// TIA Portal project "ASSEMBLER" (V16)

(* hardware
DEVICE "S7300/ET200M station_1"  S7-300 station
   slot 0: "Rail_0"  Rail  6ES7 390-1***0-0AA0
   slot 2: "PLC_1"  CPU 313C  6ES7 313-5BF03-0AB0  V2.6
      slot 0: "MPI interface_1"  X1
      slot 2: "DI 24/DO 16_1"  DI24/DO16
      slot 3: "AI 5/AO 2_1"  AI5/AO2
      slot 4: "Count_1"  Counter
*)

// ===== PLC "PLC_1"  CPU 313C =====

VAR_GLOBAL   // PLC tag table "Default tag table"
   "MOVING X" AT %I0.0 : Bool;
   "MOVING Z" AT %I0.1 : Bool;
   "ITEM DETECTED" AT %I0.2 : Bool;
   "LID AT PLACE" AT %I0.3 : Bool;
   "LID CLAMPED" AT %I0.4 : Bool;
   "POS.AT LIMIT(LIDS)" AT %I0.5 : Bool;
   "BASE AT PLACE" AT %I0.6 : Bool;
   "BASE CLAMPED" AT %I0.7 : Bool;
   "POS. AT LIMIT(BASES)" AT %I1.0 : Bool;
   "PART LEAVING" AT %I1.1 : Bool;
   "START" AT %I1.2 : Bool;
   "RESET" AT %I1.3 : Bool;
   "STOP" AT %I1.4 : Bool;
   "EMERGENCY" AT %I1.5 : Bool;
   "AUTO" AT %I1.6 : Bool;
   "MOVE X" AT %Q0.0 : Bool;
   "MOVE Z" AT %Q0.1 : Bool;
   "GRAB" AT %Q0.2 : Bool;
   "LIDS CONVEYOR" AT %Q0.3 : Bool;
   "CLAMP LID" AT %Q0.4 : Bool;
   "POS. RAISE(LID)" AT %Q0.5 : Bool;
   "BASES CONVEYOR" AT %Q0.6 : Bool;
   "CLAMP BASE" AT %Q0.7 : Bool;
   "POS. RAISE (BASES)" AT %Q1.0 : Bool;
   "START LIGHT" AT %Q1.1 : Bool;
   "RESET LIGHT" AT %Q1.2 : Bool;
   "STOP LIGHT" AT %Q1.3 : Bool;
   "COUNTER" AT %QD30 : DInt;
   "M_LID AT PLACE" AT %M0.0 : Bool;
   "stop_lid_conveyor" AT %M0.1 : Bool;
   "m_base at place" AT %M0.2 : Bool;
   "stop_base_conveyor" AT %M0.3 : Bool;
   "m_z" AT %M0.4 : Bool;
   "Run_grab" AT %M0.5 : Bool;
   "m_x" AT %M0.6 : Bool;
   "Run_x" AT %M0.7 : Bool;
   "Tag_1" AT %M1.0 : Bool;
   "set_z_after_x" AT %M1.1 : Bool;
   "Tag_2" AT %M1.2 : Bool;
   "reset grab_after x" AT %M1.3 : Bool;
   "Tag_3" AT %M1.4 : Bool;
   "set again base conveyor" AT %M1.5 : Bool;
   "Tag_4" AT %M1.6 : Bool;
   "reset system" AT %M1.7 : Bool;
   "NUMBER" AT %MD2 : DInt;
END_VAR

ORGANIZATION_BLOCK "Main"   // OB1, STL
TITLE = "Main Program Sweep (Cycle)"
{ S7_Optimized_Access := 'FALSE' }
VERSION : 0.1
   VAR_TEMP
      OB1_EV_CLASS : Byte;   // Bits 0-3 = 1 (Coming event), Bits 4-7 = 1 (Event class 1)
      OB1_SCAN_1 : Byte;   // 1 (Cold restart scan 1 of OB 1), 3 (Scan 2-n of OB 1)
      OB1_PRIORITY : Byte;   // Priority of OB Execution
      OB1_OB_NUMBR : Byte;   // 1 (Organization block 1, OB1)
      OB1_RESERVED_1 : Byte;   // Reserved for system
      OB1_RESERVED_2 : Byte;   // Reserved for system
      OB1_PREV_CYCLE : Int;   // Cycle time of previous OB1 scan (milliseconds)
      OB1_MIN_CYCLE : Int;   // Minimum cycle time of OB1 (milliseconds)
      OB1_MAX_CYCLE : Int;   // Maximum cycle time of OB1 (milliseconds)
      OB1_DATE_TIME : Date_And_Time;   // Date and time OB1 started
   END_VAR
BEGIN

REGION Network 1
         A     "START";
         O     "START LIGHT";
         A     "STOP";
         =     "START LIGHT";

         AN    "STOP";
         R     "stop_base_conveyor";
         R     "stop_lid_conveyor";
         R     "Run_grab";
         R     "Run_x";
         R     "set_z_after_x";
         R     "reset grab_after x";
         R     "POS. RAISE (BASES)";
         R     "set again base conveyor";
         R     "reset system";
END_REGION

REGION Network 2
         A     "START LIGHT";
         AN    "stop_lid_conveyor";
         =     "LIDS CONVEYOR";

         A     "START LIGHT";
         AN    "stop_base_conveyor";
         =     "BASES CONVEYOR";
END_REGION

REGION Network 3
         A     "LID AT PLACE";
         FN    "M_LID AT PLACE";
         S     "stop_lid_conveyor";

         A     "BASE AT PLACE";
         FN    "m_base at place";
         S     "stop_base_conveyor";
END_REGION

REGION Network 4
         A     "stop_lid_conveyor";
         AN    "GRAB";
         AN    "MOVE X";
         =     "CLAMP LID";

         A     "stop_base_conveyor";
         =     "CLAMP BASE";

         A     "LID CLAMPED";
         O     "set_z_after_x";
         =     "MOVE Z";

         A     "ITEM DETECTED";
         A     "MOVING Z";
         FN    "m_z";
         S     "Run_grab";

         A     "Run_grab";
         =     "GRAB";
END_REGION

REGION Network 5: RUN MOVING X
         A     "GRAB";
         A     "MOVING Z";
         FN    "m_x";
         S     "Run_x";

         A     "Run_x";
         =     "MOVE X";
END_REGION

REGION Network 6: SET MOVE Z AFTER MOVE X
         A     "GRAB";
         A     "MOVING X";
         FN    "Tag_1";
         S     "set_z_after_x";
END_REGION

REGION Network 7: RESET GRAB AFTER MOVE X
         A     "MOVE X";
         A     "MOVING Z";
         FN    "Tag_2";
         S     "reset grab_after x";


         A     "reset grab_after x";
         R     "Run_grab";
END_REGION

REGION Network 8: RESET MOVE Z \ SET PROS.(BASE) \ RESET CLAMBE BASE
         A     "MOVE X";
         AN    "GRAB";
         R     "CLAMP BASE";
         R     "set_z_after_x";
         S     "POS. RAISE (BASES)";
END_REGION

REGION Network 9: SET AGAIN BASE CONVEYOR AFTER MOVE X \ RESET stop_base_conveyor
         A     "MOVE X";
         A     "POS. AT LIMIT(BASES)";
         FN    "Tag_3";
         S     "set again base conveyor";
         R     "stop_base_conveyor";
END_REGION

REGION Network 10: RESET MOVE X \ RESET OF THE SYSTEM
         A     "PART LEAVING";
         FN    "Tag_4";
         R     "Run_x";
         R     "POS. RAISE (BASES)";
         R     "set again base conveyor";
         R     "stop_lid_conveyor";
         R     "set_z_after_x";
         R     "reset grab_after x";
         JC    INCR;
         JU    END;
END_REGION

REGION Network 11: COUNTER
   INCR: L     "NUMBER";
         L     1;
         +D;
         T     "NUMBER";

         L     "NUMBER";
         T     "COUNTER";

   END:  NOP   0;
END_REGION

REGION Network 12: RESET COUNTER
         A     "RESET";
         O     "RESET LIGHT";
         A     "STOP";
         =     "RESET LIGHT";

         A     "RESET LIGHT";
         JC    RESET;
         JU    THE_END;

   RESET:L     0;
         T     "NUMBER";
         T     "COUNTER";

   THE_END:NOP   0;
END_REGION
END_ORGANIZATION_BLOCK